/// Declaration of a distinct unit of this application
FUNCTION_BLOCK MachineUnit EXTENDS ZApplication.Unit IMPLEMENTS IMachine
VAR
  _equipment : MachineEquipment(THIS^);
  _data : MachineDataRef;
  _com : MachineComRef;

  _boot : MachineSequenceBoot(THIS^);
  _automatic : MachineSequenceAutomatic(THIS^);
  _stop : MachineSequenceStop(THIS^);
  _gohome : MachineSequenceGoHome(THIS^);
  _faultReaction : MachineSequenceFaultReaction(THIS^);
  
  _statemachine : ZApplication.UnitStateMachine;

  _observeTimer : ZAux.Timer;
END_VAR

{attribute 'ZId' := '5918240d-d585-4361-8bfb-e76d2a3c3fb9'}

_equipment.Unit.SimpleGear.PrimaryPositionC := _equipment.Unit.PrimaryGear.PrimaryPositionC;
_equipment.Unit.SimpleGear.PrimaryVelocityC := _equipment.Unit.PrimaryGear.PrimaryVelocityC;
_equipment.Unit.StruckigGear.PrimaryPositionC := _equipment.Unit.PrimaryGear.PrimaryPositionC;
_equipment.Unit.StruckigGear.PrimaryVelocityC := _equipment.Unit.PrimaryGear.PrimaryVelocityC;

IF _observeTimer.Done THEN
  _observeTimer.WaitAsync(0.1);
  
  // monitor _com for requested actions (e.g. start homing, start automatic mode, ...)
  ObserveRequest(_com.Subscribe.Request.Start, ZApplication.UnitStateMachineState.Automatic);
  ObserveRequest(_com.Subscribe.Request.Stop, ZApplication.UnitStateMachineState.Stop);
  ObserveRequest(_com.Subscribe.Request.GoHome, ZApplication.UnitStateMachineState.GoHome);
  ObserveRequest(_com.Subscribe.Request.Halt, ZApplication.UnitStateMachineState.Halt);
  
  // provide relevant information via ADS
  _com.Publish.Request.Stop := _stateMachine.IsTransitionAllowed(ZApplication.UnitStateMachineState.Stop);
  _com.Publish.Request.Start := _stateMachine.IsTransitionAllowed(ZApplication.UnitStateMachineState.Automatic);
  _com.Publish.Request.GoHome := _stateMachine.IsTransitionAllowed(ZApplication.UnitStateMachineState.GoHome);
  _com.Publish.Request.Halt := _stateMachine.IsTransitionAllowed(ZApplication.UnitStateMachineState.Halt);

  _com.Publish.State := _stateMachine.State();
END_IF

METHOD FB_init : BOOL
VAR_INPUT
  bInitRetains : BOOL; // if TRUE, the retain variables are initialized (warm start / cold start)
  bInCopyCode : BOOL;  // if TRUE, the instance afterwards gets moved into the copy code (online change)
  parent : ZCore.IManagedObject; // caller of the Unit's cyclic method. If the Unit runs in its own context use 0
  name : ZCore.ZString;  // name of this unit as it should show up in the logger
  configdata : REFERENCE TO MachineDataConfig;  // reference to the configuration data that is used during boot to configure the Units equipment
  machinedata : REFERENCE TO MachineDataMachine; // reference to the machine data that is used through most sequences of the unit (motor speed, axes positions, ...)
  calibrationdata : REFERENCE TO MachineDataCalibration;  // reference to calibration that is determined by calibration sequences of the unit (static offsets, shifts)
  com : REFERENCE TO MachineCom;  // reference to the communication interface that is used to control this Unit via ADS
END_VAR
_name := name;

// initialize local logger decorator
_loggerDecorator.FB_init(bInitRetains, bInCopyCode, name, ZModuleProgram.Logger);
_alarmingDecorator.FB_init(bInitRetains, bInCopyCode, name, ZModuleProgram.Alarming);

// setup data
_data.Config REF= configdata;
_data.Machine REF= machinedata;
_data.Calibration REF= calibrationdata;
_com.Publish REF= com.Publish;
_com.Subscribe REF= com.Subscribe;

// ------- sequence initialization, map sequences of this unit to the statemachine -------
{attribute '__ZwPlcUnitInitSequenceImplementation__'} // Do not remove this attribute! It is used for code generation.
_statemachine.SetSequence(ZApplication.UnitStateMachineState.Boot, _boot);
_statemachine.SetSequence(ZApplication.UnitStateMachineState.FaultReaction, _faultReaction);
_statemachine.SetSequence(ZApplication.UnitStateMachineState.Gohome, _gohome);
_statemachine.SetSequence(ZApplication.UnitStateMachineState.Stop, _stop);
_statemachine.SetSequence(ZApplication.UnitStateMachineState.Automatic, _automatic);

_statemachine.SetName(_name);
_statemachine.SetLogger(_logger);

// set initial state
_statemachine.SetState(ZApplication.UnitStateMachineState.Boot);
SetStateMachine(_statemachine);
END_METHOD

END_FUNCTION_BLOCK

(* stored: Version 1.1.0.1
   POU MachineUnit: Id {9b0f6c64-6abd-499c-8bc5-1e0968c49f06}, SpecialFunc None
   Folder UnitInterface: Id {4a7f1670-b05f-4e00-a802-c1b723ab9477}
   Method FB_init: Id {2eb849c2-5aa9-49e0-b41b-549c8cdadef3} *)
